// TIA Portal project "Projekt1500" (V17)

(* hardware
DEVICE "S7-1500/ET200MP-Station_1"  S7-1500 station
   slot 0: "Profilschiene_0"  Rack  6ES7 590-1***0-0AA0
   slot 1: "PLC_1"  CPU 1516-3 PN/DP  6ES7 516-3AN00-0AB0  V1.8
      slot 3: "CPU-Display_1"  6ES7591-1BA00-0AA0
      slot 32768: "PROFINET-Schnittstelle_1"  X1
         slot 32769: "Port_1"  X1 P1
         slot 32770: "Port_2"  X1 P2
      slot 33024: "PROFINET-Schnittstelle_2"  X2
         slot 33025: "Port_1"  X2 P1
      slot 33280: "DP-Schnittstelle_1"  X3
   slot 2: "DQ 32x24VDC/0.5A BA_1"  DQ 32x24VDC/0.5A BA  6ES7 522-1BL10-0AA0  V1.1
   slot 3: "DI 32x24VDC BA_1"  DI 32x24VDC BA  6ES7 521-1BL10-0AA0  V1.1
*)

// ===== PLC "PLC_1"  CPU 1516-3 PN/DP =====

VAR_GLOBAL   // PLC tag table "Standard-Variablentabelle"
   "System_Byte" AT %MB100 : Byte;
   "FirstScan" AT %M100.0 : Bool;
   "DiagStatusUpdate" AT %M100.1 : Bool;
   "AlwaysTRUE" AT %M100.2 : Bool;
   "AlwaysFALSE" AT %M100.3 : Bool;
   "Clock_Byte" AT %MB110 : Byte;
   "Clock_10Hz" AT %M110.0 : Bool;
   "Clock_5Hz" AT %M110.1 : Bool;
   "Clock_2.5Hz" AT %M110.2 : Bool;
   "Clock_2Hz" AT %M110.3 : Bool;
   "Clock_1.25Hz" AT %M110.4 : Bool;
   "Clock_1Hz" AT %M110.5 : Bool;
   "Clock_0.625Hz" AT %M110.6 : Bool;
   "Clock_0.5Hz" AT %M110.7 : Bool;
   "ASCII" AT %IB0 : Byte;   // ASCII Code des Zeichens
   "P1R" AT %Q0.0 : Bool;   // Zeiger 1 - Rechts
   "P1L" AT %Q0.1 : Bool;   // Zeiger 1 - Links
   "P2R" AT %Q0.2 : Bool;   // Zeiger 2 - Rechts
   "P2L" AT %Q0.3 : Bool;   // Zeiger 2 - Links
   "P3R" AT %Q0.4 : Bool;   // Zeiger 3 - Rechts
   "P3L" AT %Q0.5 : Bool;   // Zeiger 3 - Links
   "P4R" AT %Q0.6 : Bool;   // Zeiger 4 - Rechts
   "P4L" AT %Q0.7 : Bool;   // Zeiger 4 - Links
   "P5R" AT %Q1.0 : Bool;   // Zeiger 5 - Rechts
   "P5L" AT %Q1.1 : Bool;   // Zeiger 5 - Links
   "AlleZeiger" AT %QW0 : Word;   // Alle Zeiger
END_VAR

DATA_BLOCK "PcToPlc"   // DB1
{ S7_Optimized_Access := 'FALSE' }
VERSION : 0.1
   VAR
      Plc : Array[0..256] of Byte;
   END_VAR
BEGIN
END_DATA_BLOCK

DATA_BLOCK "PlcToPc"   // DB2
{ S7_Optimized_Access := 'FALSE' }
VERSION : 0.1
   VAR
      Plc : Array[0..256] of Byte;
   END_VAR
BEGIN
END_DATA_BLOCK

DATA_BLOCK "DeleteMe_DB"   // DB3
{ S7_Optimized_Access := 'TRUE' }
VERSION : 0.1
// stored: InstanceOfName DeleteMe
"DeleteMe"
BEGIN
END_DATA_BLOCK

FUNCTION_BLOCK "DeleteMe"   // FB1, SCL
{ S7_Optimized_Access := 'TRUE' }
VERSION : 0.1
   VAR
      Bitmuster : Array[0..256] of Word;
      Init : Bool;
      Zeiger : Int;
      Ergebnis : Word;
   END_VAR
   VAR CONSTANT
      P1R : Word := 2#0000_0000_0001;
      P1L : Word := 2#0000_0000_0010;
      P2R : Word := 2#0000_0000_0100;
      P2L : Word := 2#0000_0000_1000;
      P3R : Word := 2#0000_0001_0000;
      P3L : Word := 2#0000_0010_0000;
      P4R : Word := 2#0000_0100_0000;
      P4L : Word := 2#0000_1000_0000;
      P5R : Word := 2#0001_0000_0000;
      P5L : Word := 2#0010_0000_0000;
   END_VAR
BEGIN
   IF NOT #Init THEN
       FOR #Zeiger := 0 TO 255 DO
           #Bitmuster[#Zeiger] := 0;
       END_FOR;

       #Bitmuster[16#41] := #P1R + #P5L; //65 A
       #Bitmuster[16#42] := #P1R + #P4L; //66 B
       #Bitmuster[16#44] := #P2R + #P5L; //68 D
       #Bitmuster[16#45] := #P1R + #P3L; //69 E
       #Bitmuster[16#46] := #P2R + #P4L; //70 F
       #Bitmuster[16#47] := #P3R + #P5L; //71 G
       #Bitmuster[16#48] := #P1R + #P2L; //72 H
       #Bitmuster[16#49] := #P2R + #P3L; //73 I
       #Bitmuster[16#4B] := #P3R + #P4L; //75 K
       #Bitmuster[16#4C] := #P4R + #P5L; //76 L

       #Bitmuster[16#4D] := #P1L + #P2R; //77 M
       #Bitmuster[16#4E] := #P2L + #P3R; //78 N
       #Bitmuster[16#4F] := #P3L + #P4R; //79 O
       #Bitmuster[16#50] := #P4L + #P5R; //80 P
       #Bitmuster[16#52] := #P1L + #P3R; //82 R
       #Bitmuster[16#53] := #P2L + #P4R; //83 S
       #Bitmuster[16#54] := #P3L + #P5R; //84 T
       #Bitmuster[16#56] := #P1L + #P4R; //86 V
       #Bitmuster[16#57] := #P2L + #P5R; //87 W
       #Bitmuster[16#59] := #P1L + #P5R; //89 Y    
   END_IF;

   #Ergebnis := #Bitmuster["ASCII"];

   POKE(area := 16#84, dbNumber := 1, byteOffset := 0, value := #Ergebnis.%B0);
   POKE(area := 16#84, dbNumber := 1, byteOffset := 1, value := #Ergebnis.%B1);
END_FUNCTION_BLOCK

FUNCTION "DatenRangieren" : Void   // FC1, SCL
{ S7_Optimized_Access := 'TRUE' }
VERSION : 0.1
   VAR_TEMP
      TextLaenge : UInt;
   END_VAR
BEGIN
   // Area 16#81 --> Input
   // Area 16#82 --> Output
   // Area 16#84 --> DB

   POKE(area := 16#81,                     // DI (Hardware PLC)
        dbNumber := 0,
        byteOffset := 0,
        value := PEEK(area := 16#84, dbNumber := 1, byteOffset := 0));


   Strg_TO_Chars(Strg := 'Nadeltelegraph V3.0',
                 pChars := 96,
                 Cnt=>#TextLaenge,
                 Chars := "PlcToPc".Plc);
END_FUNCTION

ORGANIZATION_BLOCK "Main"   // OB1, LAD, ProgramCycle
TITLE = "Main Program Sweep (Cycle)"
{ S7_Optimized_Access := 'TRUE' }
VERSION : 0.1
   VAR_INPUT
      Initial_Call : Bool;   // Initial call of this OB
      Remanence : Bool;   // =True, if remanent data are available
   END_VAR
BEGIN

REGION Network 1
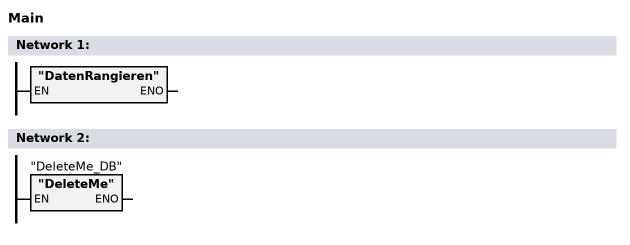
   RUNG wire#powerrail
      "DatenRangieren"()
   END_RUNG
   // the same network as SCL:
   "DatenRangieren"();
END_REGION

REGION Network 2
   RUNG wire#powerrail
      "DeleteMe_DB"()
   END_RUNG
   // the same network as SCL:
   "DeleteMe_DB"();   // "DeleteMe"
END_REGION
END_ORGANIZATION_BLOCK

ORGANIZATION_BLOCK "Startup"   // OB100, SCL, Startup
TITLE = "Complete Restart"
{ S7_Optimized_Access := 'TRUE' }
VERSION : 0.1
   VAR_INPUT
      LostRetentive : Bool;   // True if retentive data are lost
      LostRTC : Bool;   // True if date and time are lost
   END_VAR
BEGIN
   // Area 16#81 --> Input
   // Area 16#82 --> Output
   // Area 16#84 --> DB

   POKE(area := 16#82, dbNumber := 0, byteOffset := 0, value := byte#0);  // Ausgänge löschen
END_ORGANIZATION_BLOCK